FUNCTION_BLOCK FB_EventHandler EXTENDS FB_Handler
VAR_INPUT
END_VAR
VAR_OUTPUT
	bDebug:			BOOL;
	bInfo:			BOOL;
	bWarning:		BOOL;
	bError:			BOOL;
END_VAR
VAR
	nLength:		INT;
	aEvents:		ARRAY [0..100] OF ST_Event;
	nIndex: 		INT;
END_VAR

SUPER^();
nIndex:= 0;
WHILE nIndex < nLength DO
	IF aEvents[nIndex].bActive THEN
		aEvents[nIndex].bActive:= FALSE;
	ELSE
		M_Remove(nIndex);
	END_IF
	nIndex := nIndex + 1;
END_WHILE
bDebug:= FALSE;
bInfo:= FALSE;
bWarning:= FALSE;
bError:= FALSE;

METHOD PRIVATE M_Find : INT
VAR_INPUT
	stEvent:			ST_Event;		// event to find
END_VAR
M_Find := -1;
nIndex:= 0;
WHILE nIndex < nLength DO
    IF aEvents[nIndex].eEvent = stEvent.eEvent AND_THEN aEvents[nIndex].sMessage = stEvent.sMessage THEN
        M_Find := nIndex;
        RETURN;
    END_IF
	nIndex := nIndex + 1;
END_WHILE
END_METHOD

METHOD PRIVATE M_Remove
VAR_INPUT
	nPosition:			INT;
END_VAR
memcpy(ADR(aEvents[nIndex]), ADR(aEvents[nPosition + 1]), (SIZEOF(ST_Event) * (100  - nPosition)));
nLength:= nLength - 1;
END_METHOD

METHOD PUBLIC M_Request
VAR_INPUT
	stEvent:			ST_Event;		// event to be handled. 
END_VAR
VAR
	nFind:				INT;
END_VAR
IF nLength < 100 THEN
	nFind:= M_Find(stEvent);
	IF nFind = -1 THEN
		aEvents[nLength]:= stEvent;
		nLength:= nLength + 1;
	ELSE
		aEvents[nFind]:= stEvent;
		CASE aEvents[nFind].eEvent OF
			E_Event.Debug:
				bDebug:= TRUE;
			E_Event.Info:
				bInfo:= TRUE;
			E_Event.Warning:
				bWarning:= TRUE;
			E_Event.Error:
				bError:= TRUE;
		END_CASE
		
	END_IF
END_IF

SUPER^.M_Request(stEvent);
END_METHOD

END_FUNCTION_BLOCK

(* stored: Version 1.1.0.1, ProductVersion 3.1.4024.12
   POU FB_EventHandler: Id {a7ae2211-d1a6-49e2-82c8-5c610d8a7c9d}, SpecialFunc None
   Method M_Find: Id {bb4df97c-6e38-4cd5-bdfc-6c0b84052df0}
   Method M_Remove: Id {78bc2cb4-2b52-4154-8478-d32962040d8c}
   Method M_Request: Id {fd7a157e-fd8c-45f8-a7bc-2309e3dc7519} *)
